PROGRAM PRG_Test
VAR
	isInRangeFunctionsTest : IsInRangeInclusiveFunctionsTest;
END_VAR

TcUnit.RUN();

END_PROGRAM

(* stored: Version 1.1.0.1, ProductVersion 3.1.4024.15
   POU PRG_Test: Id {5869bc1e-7216-0262-2153-7c31dd278f58}, SpecialFunc None *)
